(* IEC 61131-3 sources: test_training/GmpAccess2/src/Functionblocks, 2 files *)

(* ---- Calculator.st ---- *)
FUNCTION_BLOCK Calculator
VAR_INPUT
	in1 : REAL;
	in2 : REAL;
END_VAR

VAR_OUTPUT
	out : REAL;
END_VAR

VAR

END_VAR

add1;
sub1;
mul1;
div1;

END_FUNCTION_BLOCK

ACTIONS

ACTION add1
	out := in1 + in2;
END_ACTION

ACTION sub1
	out := in1 - in2;
END_ACTION

ACTION mul1
	out := in1 * in2;
END_ACTION

ACTION div1
	out := in1 / in2;
END_ACTION

END_ACTIONS

(* ---- ChanValue.st ---- *)
FUNCTION_BLOCK ChanValue
VAR_INPUT
	value AT %I*: DWORD;
	i : INT;
END_VAR

VAR_OUTPUT

END_VAR

VAR

END_VAR

VoltageL1x_TRMS_HCC;
VoltageL2x_TRMS_HCC;
VoltageL3x_TRMS_HCC;
i := i + 1;
END_FUNCTION_BLOCK
